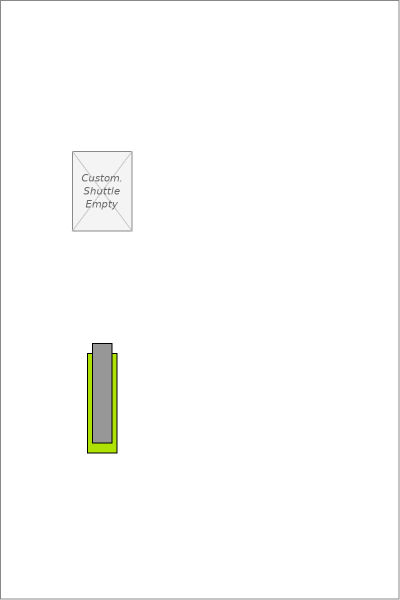
VISUALIZATION VISU_ST170  // 400x600
    Image (72,151 60x80), angle 90, invisible if: NOT __ISVALIDREF(GVL.st170_aut._Mover), image: Custom.Shuttle Empty
    Rectangle (87,353 30x100)
    Rectangle (92,343 20x100)
        p2738717112: -GVL.st170_aut.fb_ABL_RFID.simu_axis170_01Z.rOUT_PixActual
END_VISUALIZATION

(* stored: Version 1.1.0.1, ProductVersion 3.1.4024.6
   Visu VISU_ST170: Id {efa6f6c5-9216-4f42-8309-8db7efb92aec} *)
